FUNCTION_BLOCK FB_CONVEYANCE
VAR_INPUT
END_VAR
VAR_OUTPUT
END_VAR
VAR
END_VAR

END_FUNCTION_BLOCK

(* stored: Version 1.1.0.1, ProductVersion 3.1.4024.12
   POU FB_CONVEYANCE: Id {7bebbc7a-8549-4ab0-9f56-d4d12bd0462a}, SpecialFunc None *)
